Staubli VAL3: secuTask1.pgx

public program secuTask1()
// Control "Mould Area Free" from robot
  local point pLocFlange
  local point pLocTCP
begin
  //
  //!change 23.04.06, vdg: added global variable that contains the distance to the safety zone
  // Security zon in millimeter for wrist relativ to IMM Backside...........
  // nSafeZon[0]=300
  //
  // LOOP: task "RobSafe1"..................................................

    //
    // Get current robot position relative to the frame of IMM Backside.....
    pLocFlange=here(flange,data:fAreaIMM)
    pLocTCP=here(data:tTCP,data:fAreaIMM)
    //
    // Set signal "Mould Area Free" to machine..............................
    nMouldAreaDist=max(pLocTCP.trsf.z,pLocFlange.trsf.z)-nMouldAreaZone
    SYS:doMouldFree[moduleIndex]=nMouldAreaDist<0
    //
    if SYS:doMouldFree==false
      SYS:doStartMachine=false
      bRobotOff=false
    endIf
    //
    //!change 18.05.06, vdg: Test if MouldFree Signal has toggled while robot was in mould
    switch nAreaTestState
      // initialize test
      case 0
        //nAreaTestState=0
        //bAreaFlag=SYS:doMouldFree
      break
      // wait for high state
      case 10
        if SYS:doMouldFree==true
          nAreaTestState=20
        endIf
      break
      // wait for low state
      case 20
        if SYS:doMouldFree==false
          nAreaTestState=30
        endIf
      break
      // wait for high state again
      case 30
        if SYS:doMouldFree==true
          nAreaTestState=40
        endIf
      break
      // final state
      // this state must be reached when startIMM() is called
      case 40
      break
    endSwitch
//  SYS:doSecu[0]=false
//  SYS:doSecu[1]=false
end
